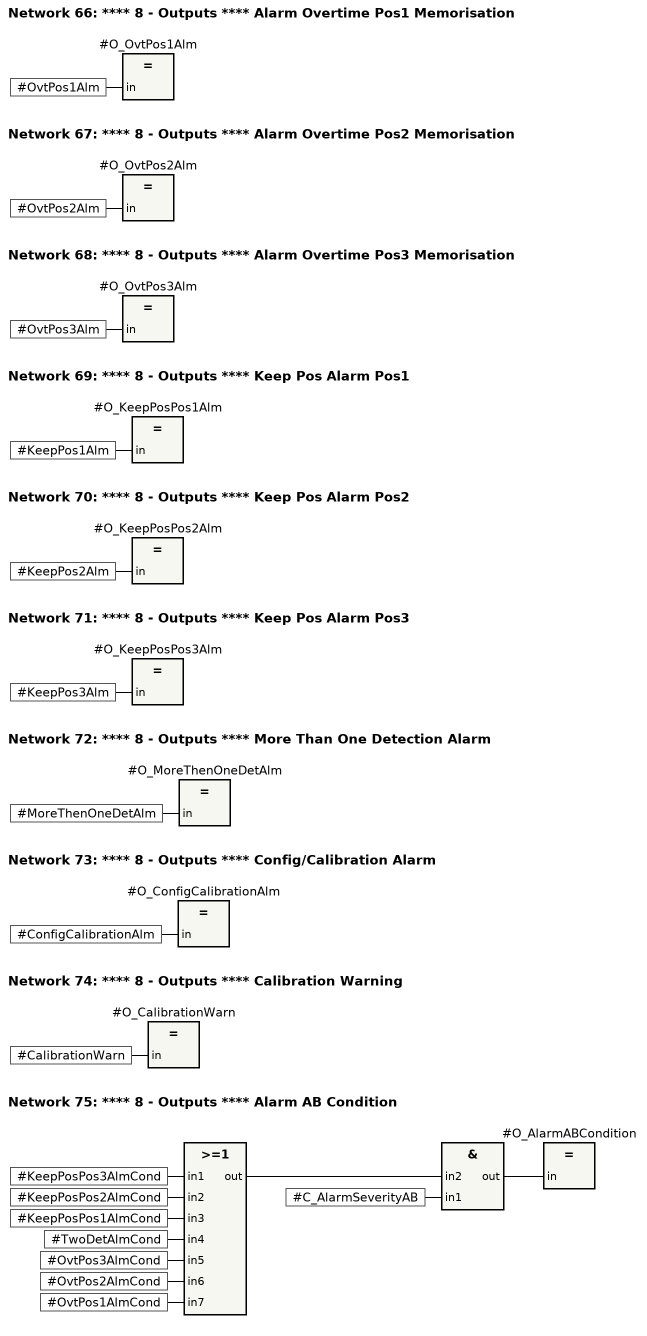
   #O_OvtPos1Alm := #OvtPos1Alm;
END_REGION

REGION Network 67: **** 8 - Outputs **** Alarm Overtime Pos2 Memorisation
   // Alarm Overtime Pos2 Memorisation
   #O_OvtPos2Alm := #OvtPos2Alm;
END_REGION

REGION Network 68: **** 8 - Outputs **** Alarm Overtime Pos3 Memorisation
   // Alarm Overtime Pos3  Memorisation
   #O_OvtPos3Alm := #OvtPos3Alm;
END_REGION

REGION Network 69: **** 8 - Outputs **** Keep Pos Alarm Pos1
   // Keep Pos Alarm Pos1
   #O_KeepPosPos1Alm := #KeepPos1Alm;
END_REGION

REGION Network 70: **** 8 - Outputs **** Keep Pos Alarm Pos2
   // Keep Pos Alarm Pos2
   #O_KeepPosPos2Alm := #KeepPos2Alm;
END_REGION

REGION Network 71: **** 8 - Outputs **** Keep Pos Alarm Pos3
   // Keep Pos Alarm Pos3
   #O_KeepPosPos3Alm := #KeepPos3Alm;
END_REGION

REGION Network 72: **** 8 - Outputs **** More Than One Detection Alarm
   // More Than One Detection Alarm
   #O_MoreThenOneDetAlm := #MoreThenOneDetAlm;
END_REGION

REGION Network 73: **** 8 - Outputs **** Config/Calibration Alarm
   #O_ConfigCalibrationAlm := #ConfigCalibrationAlm;
END_REGION

REGION Network 74: **** 8 - Outputs **** Calibration Warning
   #O_CalibrationWarn := #CalibrationWarn;
END_REGION

REGION Network 75: **** 8 - Outputs **** Alarm AB Condition
   // Alarm AB Condition
   #O_AlarmABCondition := (#KeepPosPos3AlmCond OR #KeepPosPos2AlmCond OR #KeepPosPos1AlmCond OR #TwoDetAlmCond OR #OvtPos3AlmCond OR #OvtPos2AlmCond OR #OvtPos1AlmCond) AND #C_AlarmSeverityAB;
END_REGION
END_FUNCTION_BLOCK
